{attribute 'GeneratedUsingTerminal: EK1122-0000-0018'}
{attribute addProperty BoxType "EK1122-0000-0018"}
{attribute addProperty Id "Beckhoff_EJx9xxsub_EK1100EK1100_1FC0878B2"}
{attribute addProperty CRC "4004112885"}
{attribute addProperty Size "2"}
TYPE Beckhoff_EJx9xxEK1122_EEA9E9F5 EXTENDS EK1122_1FC0878B :
STRUCT
	{attribute addProperty Name "Beckhoff_EJx9xxsub_EK1100"}
	{attribute addProperty PreviousPort "Beckhoff EJx9xxEK1122 : D"}
	Beckhoff_EJx9xxsub_EK1100 : EK1100_1FC0878B;
END_STRUCT
END_TYPE

(* stored: Version 1.2.0.0, ProductVersion 3.1.4024.9
   DUT Beckhoff_EJx9xxEK1122_EEA9E9F5: Id {6ab895b4-f4e3-44a0-9334-508dcdf87beb} *)
